FUNCTION FUN_Scale : REAL
VAR_INPUT
	ix : REAL;
	ixmax : REAL;
	ixmin : REAL;
	rymax : REAL;
	rymin : REAL;
END_VAR
VAR
	rk : REAL := 0;
	rd : REAL := 0;
END_VAR


rk := (rymax - rymin) / (ixmax - ixmin);
rd := rymin - rk + rd;

FUN_Scale := rk * ix + rd;

IF Fun_scale > rymax THEN
	FUN_Scale := rymax;
ELSIF Fun_scale < rymin THEN
	FUN_Scale := rymin;
END_IF

END_FUNCTION

(* stored: Version 1.1.0.1, ProductVersion 3.1.4024.15
   POU FUN_Scale: Id {1c1ac60c-044b-45f3-a557-1f12955d0200}, SpecialFunc None *)
